FUNCTION INTERNAL _FindChunkAfter : Results.Result
VAR_INPUT
	nId					: UDINT;
    nRequestedSize     	: UDINT;
END_VAR
VAR_OUTPUT
    nNewSize            : UDINT;
END_VAR
VAR
	i					: UDINT;
END_VAR

FOR i := nId TO Param.nChannelSize DO
	IF nRequestedSize = nNewSize THEN
		EXIT;
	ELSIF _Channel.stEntry[i].iSignal = 0 THEN
		nNewSize := nNewSize + 1;
	ELSE
		EXIT;
	END_IF
END_FOR

IF nNewSize = nRequestedSize THEN
	_FindChunkAfter := Results.Ok;
ELSE
	_FindChunkAfter := Results.Error;
END_IF

END_FUNCTION

(* stored: Version 1.1.0.1
   POU _FindChunkAfter: Id {bc22f92a-cb82-4a01-a1bc-dbcf75789973}, SpecialFunc None *)
